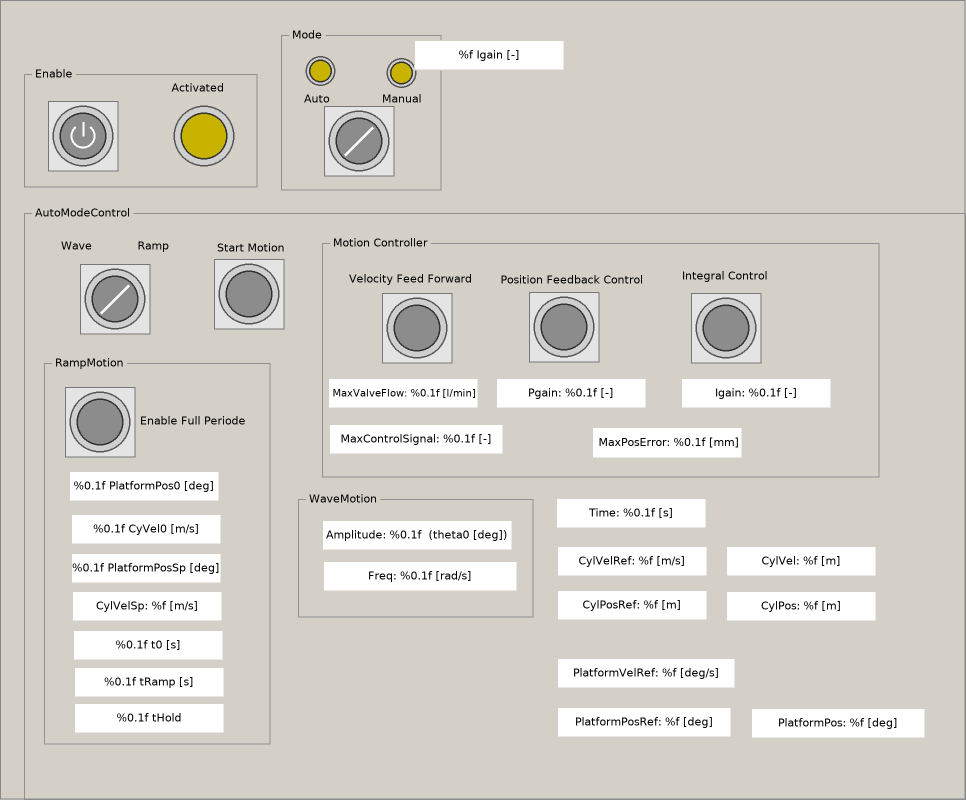
VISUALIZATION StablePlatform  // 966x800
    GroupBox (281,27 160x163), "Mode"
        RotarySwitch (43,79 70x70), variable: G_StablePlatformIO.bModeSelector, behaviour: TOGGLE, style: Switch-RotarySwitch-Gray
        Lamp1 (21,27 37x34), variable: G_StablePlatformIO.bAutoMode, style: Lamp-Lamp1-Yellow
        Lamp1 (102,29 37x34), variable: G_StablePlatformIO.bManualMode, style: Lamp-Lamp1-Yellow
        Label (7,57 150x30), "Auto Manual"
    GroupBox (24,66 233x121), "Enable"
        PowerSwitch (24,35 70x70), variable: G_StablePlatformIO.bEnable, behaviour: TOGGLE, style: Switch-PowerSwitch-Gray
        Lamp1 (145,35 70x70), variable: G_StablePlatformIO.bActivated, style: Lamp-Lamp1-Yellow
    GroupBox (24,205 942x595), "AutoModeControl"
        RotarySwitch (56,59 70x70), variable: G_StablePlatformIO.bMotionModeSelector, behaviour: TOGGLE, style: Switch-RotarySwitch-Gray
        Label (16,26 150x30), "Wave Ramp"
        PushSwitch (190,54 70x70), variable: G_StablePlatformIO.bStartMotionGenerator, behaviour: TOGGLE, style: Switch-PushSwitch-Gray
        Label (152,28 150x30), "Start Motion"
        GroupBox (20,150 226x389), "RampMotion"
            PushSwitch (21,32 70x70), variable: G_StablePlatformIO.bRampMotionFullPeriode, behaviour: TOGGLE, style: Switch-PushSwitch-Gray
            Label (74,51 150x30), "Enable Full Periode"
            Textfield (25,116 150x30), "%0.1f PlatformPos0 [deg]", text variable: G_StablePlatformIO.bRampMotionPos0_deg
                OnMouseDown: write the text variable via Default
            Textfield (27,159 150x30), "%0.1f CyVel0 [m/s]", text variable: G_StablePlatformIO.bRampMotionCylVel0_ms
                OnMouseDown: write the text variable via Default
            Textfield (27,198 150x30), "%0.1f PlatformPosSp [deg]", text variable: G_StablePlatformIO.bRampMotionPositionSP_deg
                OnMouseDown: write the text variable via Default
            Textfield (28,236 150x30), "CylVelSp: %f [m/s]", text variable: G_StablePlatformIO.bRampMotionVelocitySP_ms
                OnMouseDown: write the text variable via Default
            Textfield (29,275 150x30), "%0.1f t0 [s]", text variable: G_StablePlatformIO.bRampMotiont0_s
                OnMouseDown: write the text variable via Default
            Textfield (30,312 150x30), "%0.1f tRamp [s]", text variable: G_StablePlatformIO.bRampMotiontRamp_s
                OnMouseDown: write the text variable via Default
            Textfield (30,348 150x30), "%0.1f tHold", text variable: G_StablePlatformIO.bRampMotiontHoldPos_s
                OnMouseDown: write the text variable via Default
        Textfield (532,293 150x30), "Time: %0.1f [s]", text variable: G_StablePlatformIO.fTime
        GroupBox (274,286 235x126), "WaveMotion"
            Textfield (24,29 190x30), "Amplitude: %0.1f (theta0 [deg])", text variable: G_StablePlatformIO.fWaveMotionAplitudeTheta0_deg
                OnMouseDown: write the text variable via Default
            Textfield (25,70 194x30), "Freq: %0.1f [rad/s]", text variable: G_StablePlatformIO.WaveMotionFreq_rads
                OnMouseDown: write the text variable via Default
        Textfield (533,341 150x30), "CylVelRef: %f [m/s]", text variable: G_StablePlatformIO.fCylVelRef_ms
        Textfield (533,385 150x30), "CylPosRef: %f [m]", text variable: G_StablePlatformIO.fCylPosRef_m
        Textfield (702,386 150x30), "CylPos: %f [m]", text variable: G_StablePlatformScaledIO.fPistonPosition
        Textfield (702,341 150x30), "CylVel: %f [m]", text variable: G_StablePlatformScaledIO.fPistonVelocity
        Textfield (533,453 178x30), "PlatformVelRef: %f [deg/s]", text variable: G_StablePlatformIO.fWaveMotionOmega_degs
        Textfield (533,502 174x30), "PlatformPosRef: %f [deg]", text variable: G_StablePlatformIO.fWaveMotionTheta_deg
        Textfield (727,503 174x30), "PlatformPos: %f [deg]", text variable: G_StablePlatformScaledIO.fPlatformAngleDeg
        Textfield (390,-165 150x30), "%f Igain [-]", text variable: G_StablePlatformIO.fIntegralGain
        GroupBox (298,30 557x242), "Motion Controller"
            PushSwitch (60,58 70x70), variable: G_StablePlatformIO.bEnableFeedForward, behaviour: TOGGLE, style: Switch-PushSwitch-Gray
            PushSwitch (207,57 70x70), variable: G_StablePlatformIO.bEnableFeedBackControl, behaviour: TOGGLE, style: Switch-PushSwitch-Gray
            PushSwitch (369,58 70x70), variable: G_StablePlatformIO.bEnableIntegralControl, behaviour: TOGGLE, style: Switch-PushSwitch-Gray
            Textfield (270,192 150x31), "MaxPosError: %0.1f [mm]", text variable: G_StablePlatformIO.fMaxPosError_mm
                OnMouseClick: write the text variable via Default
            Textfield (174,143 150x30), "Pgain: %0.1f [-]", text variable: G_StablePlatformIO.fProportionalGain
                OnMouseClick: write the text variable via Default, min 0.0000001
            Textfield (6,143 150x30), "MaxValveFlow: %0.1f [l/min]", text variable: G_StablePlatformIO.fMaxValveFlow_lmin
                OnMouseClick: write the text variable via Default
            Textfield (359,143 150x30), "Igain: %0.1f [-]", text variable: G_StablePlatformIO.fIntegralGain
                OnMouseClick: write the text variable via Default
            Label (175,30 150x30), "Position Feedback Control"
            Label (328,26 150x30), "Integral Control"
            Textfield (7,189 174x30), "MaxControlSignal: %0.1f [-]", text variable: G_StablePlatformParameters.fMaxControlSignal
                OnMouseClick: write the text variable via Default, min -1, max 1
        Label (297,59 179x30), "Velocity Feed Forward"
    Label (123,73 150x30), "Activated"
END_VISUALIZATION

(* stored: Version 1.1.0.1, ProductVersion 3.1.4024.12
   Visu StablePlatform: Id {948dac3a-1fd6-4fe6-86cb-5e13c0e37bad} *)
